Universal Robots PolyScope program: robotprogfirst.urp

Program robotprogfirst (installation=default directory=/programs/usbdisk_1/URscript createdIn=3.9.1.64192 lastSavedIn=3.9.1.64192 robotSerialNumber=2016331617)
Calibrated DH parameters: a=[-0.000045, -0.22956, -0.153032, 0.000019, 0.0001, 0]; d=[0.152163, -856.35044, 904.692211, -48.229373, 0.085425, 0.082565]; alpha=[1.571202, -0.000097, 0.003084, 1.571016, -1.571253, 0]; deltaTheta=[-0.00003, 0.346154, 0.426056, -0.772366, 0.00006, 0.000029]
BeforeStart
  Script: conres = socket_open("192.168.137.1",23)
  Script: textmsg(conres)
  Script: targetPos=p[0, 0, 0, 0, 0, 0]
  Script: receiveFromServ=[0, 0, 0, 0, 0, 0, 0, 0]
Robot Program (runOnlyOnce=false)
  Script: sendToServer="Klar"
  Script: socket_send_string(sendToServer)
  Loop While (checkContinuously=false) expression=conres≟ True
    Script: receiveFromServ=socket_read_ascii_float(7)
    Script: textmsg(receiveFromServ)
    If receiveFromServ[7]≟1
      Script: break
    ElseIf receiveFromServ[7]≟2
      Script: break
    ElseIf receiveFromServ[7]≟3
      Script: break
    ElseIf receiveFromServ[7]≟4
      Script: break
  Loop Forever
    Script: targetPos=p[receiveFromServ[1],receiveFromServ[2],receiveFromServ[3],receiveFromServ[4],receiveFromServ[5],receiveFromServ[6]]
    Script: textmsg(targetPos)
    If targetPos≠p[0, 0, 0, 0, 0, 0]
      MoveL speed 250 mm/s, acceleration 1200 mm/s^2 (useActiveTCP=true) feature=Base
        Waypoint Waypoint (Variable): variable=targetPos
      Script: break
  SuppressedNode
    Loop While (checkContinuously=false) expression=receiveFroomServ[0]≠6
      Wait Sleep waitTime=0.3
      Script: receiveFromServ=socket_read_ascii_float(6)
  Wait Sleep waitTime=1
  Script: targetPos=p[0, 0, 0, 0, 0, 0]
  MoveL speed 250 mm/s, acceleration 1200 mm/s^2 (useActiveTCP=true) feature=Base
    Waypoint Waypoint_1: TCP in base x=-218.947 y=103.634 z=576.492 mm, rx=-0.8555 ry=-1.2749 rz=-0.1412 rad; joints [-62.287, -105.827, 77.47, -154.059, -66.74, -60.096] deg
